FUNCTION_BLOCK ABSTRACT IonizerBase EXTENDS TExecution IMPLEMENTS IDevice
VAR_INPUT
END_VAR
VAR_OUTPUT
END_VAR
VAR
	{attribute 'OPC.UA.DA' := '0'}
	_name : STRING;
	{attribute 'OPC.UA.DA' := '0'}
	_deviceID : STRING;				
	{attribute 'OPC.UA.DA' := '0'}
	_family : DeviceFamily := DeviceFamily.Ionizer;		
	{attribute 'OPC.UA.DA' := '0'}
	_logger : Logger;
	{attribute 'OPC.UA.DA' := '0'}
	_message : StringBuilder;
	{attribute 'OPC.UA.DA' := '0'}
	_ionizerConfig : DeviceConfiguration;
		
	{attribute 'OPC.UA.DA' := '0'}
	_lifeTimeCount : UINT;
	{attribute 'OPC.UA.DA' := '0'}
	_notifyIsAlive : BOOL;
	{attribute 'OPC.UA.DA' := '0'}
	_pulseIsAliveGenerator : TON;

	StateMsg : STRING(255);
	IsAliveMsg : STRING(255);
END_VAR

// Check if it's still alive	
IF _notifyIsAlive THEN
	IsAliveMsg := TO_STRING(_lifeTimeCount);
	_notifyIsAlive := FALSE;
END_IF

IF HardwareGlobalVariables.IonizerState <> State THEN
	HardwareGlobalVariables.IonizerState := State;
	StateMsg := ANY_TO_STRING(State);		
END_IF

PROPERTY DeviceID : STRING
GET
DeviceID := _deviceID;
END_GET
SET
_deviceID := DeviceID;
END_SET
END_PROPERTY

PROPERTY Family : DeviceFamily
GET
Family := _family;
END_GET
SET
_family := Family;
END_SET
END_PROPERTY

METHOD PROTECTED IsAlive
VAR_INPUT
END_VAR
_notifyIsAlive := TRUE;

IF _lifeTimeCount < 5 THEN
	_lifeTimeCount := _lifeTimeCount + 1;
ELSE
	_lifeTimeCount := 1;
END_IF
END_METHOD

PROPERTY Name : STRING
GET
Name := _name;
END_GET
SET
_name := Name;
END_SET
END_PROPERTY

END_FUNCTION_BLOCK

(* stored: Version 1.1.0.1, ProductVersion 3.1.4024.12
   POU IonizerBase: Id {9120f6c9-f01f-4c66-9084-edbe42ad7f1b}, SpecialFunc None
   Folder Commands: Id {da1cedff-f136-4578-9360-cf11b5b8c801}
   Property DeviceID: Id {200c18b4-daa2-487b-87c4-560f294111a5}
   Get Get: Id {ccb139d9-37ee-496a-94da-1c99ddb32288}
   Set Set: Id {7df119ab-3077-4432-8339-77f7d69017fc}
   Property Family: Id {55e7a5e2-87ba-4bdd-8fdd-83591c567fcb}
   Get Get: Id {f9371fe8-aa34-434c-9653-11b54b1d9c31}
   Set Set: Id {faabad28-2bfa-48d5-a366-66ce15c55c3e}
   Method IsAlive: Id {eb2cfc23-65bc-498b-8440-38437a0d4457}
   Property Name: Id {cb90871f-163d-4ae0-9785-57cae66ea028}
   Get Get: Id {7d066735-d742-4c0d-8e15-0f664a8c3ca1}
   Set Set: Id {d3e22868-f5a2-4efa-bcd0-79edf270bf84} *)
